INTERFACE I_LedDevice EXTENDS I_Display

METHOD PUBLIC ConnectTo
VAR_INPUT
	LedDevice : I_LedDevice;
END_VAR
END_METHOD

METHOD PUBLIC ResetPixelPointer
VAR_INPUT
END_VAR
END_METHOD

METHOD PUBLIC TryGetNextPixel : BOOL
VAR_INPUT
	Destination : REFERENCE TO Pixel;
END_VAR
END_METHOD

METHOD PUBLIC UpdateFrom
VAR_INPUT
	Source : I_ReadableDisplayBuffer;
END_VAR
END_METHOD

END_INTERFACE

(* stored: Version 1.1.0.1, ProductVersion 3.1.4024.15
   Itf I_LedDevice: Id {1b8cc47e-34ff-499b-a9f6-4d022b370077}
   Method ConnectTo: Id {3d386719-ae8c-4d9c-b65d-39f64c511c37}
   Method ResetPixelPointer: Id {cd438b9f-08ba-43c1-a34f-98d5f639752a}
   Method TryGetNextPixel: Id {21e43cb1-5489-43b4-bcc6-bf578ada4c16}
   Method UpdateFrom: Id {84894468-cbaf-43ca-af9a-680ff605d81b} *)
